// TIA Portal V18 export
// export: Created 2026-03-12T16:04:35.9401057Z, ExportSetting WithDefaults, DisplayName Totally Integrated Automation Portal, DisplayVersion V18 Update 5, DisplayName TIA Portal Openness, DisplayVersion V18 Update 5, DisplayName TIA Portal Version Control Interface, DisplayVersion V18, DisplayName SINAMICS Startdrive Advanced, DisplayVersion V18, DisplayName SINAMICS Startdrive G130, G150, S120, S150, SINAMICS MV, S210, DisplayVersion V18, DisplayName SINAMICS Startdrive G110M, G120, G120C, G120D, G120P, G115D, DisplayVersion V18, DisplayName STEP 7 Professional, DisplayVersion V18 Update 5, DisplayName STEP 7 Safety, DisplayVersion V18, DisplayName WinCC Professional, DisplayVersion V18 Update 5
FUNCTION_BLOCK "FB_INICIADOR_COMM_SKID"   // FB29, SCL
{ S7_Optimized_Access := 'TRUE' }
VERSION : 0.1
// stored: AutoNumber true, IsIECCheckEnabled false, IsRetainMemResEnabled false, MemoryReserve 100, SetENOAutomatically false, UDAEnableTagReadback false
   VAR_INPUT
      HABILITA : Bool;
      DONE : Bool;
      BUSY : Bool;
      STATUS_WORD : Word;
      tCTU : Time := T#20s;
      tBUSY : Time;
      id_Max : Word := 10;
   END_VAR
   VAR_OUTPUT
      ERROR : Bool;
   END_VAR
   VAR_IN_OUT
      Tcom_IP_4 : TCON_IP_v4;
      Conected : Bool;
   END_VAR
   VAR
      FIRST_RUN : Bool := TRUE;
      tWait_Ctu : TON_TIME;
      tWait_Ctu_1 { S7_SetPoint := 'True'} : TON_TIME;
      tWait_Busy { S7_SetPoint := 'True'} : TON_TIME;
      Status_OK { S7_SetPoint := 'True'} : Bool;
      index : Int;
   END_VAR
BEGIN
   (* // =======================
   // LÓGICA PRINCIPAL
   // =======================
   IF not #HABILITA THEN
       #tWait_Ctu.IN := FALSE;
       #tWait_Busy.IN := FALSE;
       RETURN;
   END_IF;


   // =======================
   // STATUS VÁLIDOS
   // =======================
   #Status_OK := (#STATUS_WORD = 16#0000) OR
   (#STATUS_WORD = 16#0001) OR
   (#STATUS_WORD = 16#7000) OR
   (#STATUS_WORD = 16#7004) OR
   (#STATUS_WORD = 16#7005) OR
   (#STATUS_WORD = 16#7006);


   // =======================
   // MONITORA BUSY
   // =======================
   #tWait_Busy(IN := #BUSY,   PT := #tBUSY);

   // =======================
   // PRIMEIRA EXECUÇÃO
   // =======================
   IF #FIRST_RUN THEN
       #index := 1;
       #Tcom_IP_4.ID := INT_TO_WORD(#index);
       #FIRST_RUN := FALSE;
   END_IF;


   // =======================
   // CONDIÇÃO DE SUCESSO
   // =======================
   IF #DONE AND #Status_OK AND NOT #tWait_Busy.Q THEN
       // Comunicação consolidada
       #index := 1;
       #Tcom_IP_4.ID := INT_TO_WORD(#index);

       #tWait_Ctu.IN := FALSE;
       #tWait_Busy.IN := FALSE;
       #ERROR := FALSE;

       // =======================
       // MODO SCAN 
       // =======================
   ELSE
       #ERROR := TRUE;

       // Só entra em varredura se BUSY travou ou DONE não confirmou
       IF #tWait_Busy.Q OR NOT #DONE THEN
           #tWait_Ctu(IN := TRUE,  PT := #tCTU);
           #tWait_Ctu_1(IN := NOT #Conected,
                      PT := #tCTU);
         #Conected := #tWait_Ctu_1.Q;

           IF #tWait_Ctu.Q THEN
               #index := #index + 1;

               IF #index > #id_Max THEN
                   #index := 1;
               END_IF;

               #Tcom_IP_4.ID := INT_TO_WORD(#index);
               #tWait_Ctu.IN := FALSE; // rearma ciclo

           END_IF;

           #tWait_Ctu_1.IN := FALSE; // rearma ciclo
       END_IF;
   END_IF;
   *)
END_FUNCTION_BLOCK
